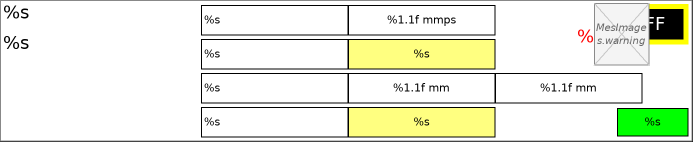
VISUALIZATION VISU_AXE_STD1_LIN_REL_FCT_ETAT_OSC  // 693x142
VAR_IN_OUT
	m_Input_MOTEUR: BLOCK_AXE_STD1_OSCILLANT;
	m_Input_PRG_MOUVEMENT_PS: BLOCK_PRG_MOUVEMENT_PS;
END_VAR
VAR_INPUT
	m_Input_ID_NOM_XML : INT;
END_VAR
    Rectangle (0,0 693x142), "%s", text list: 'TextList_Type_Moteur', text index: m_Input_ID_NOM_XML
    Rectangle (0,28 107x30), "%s", text variable: m_Input_MOTEUR.MNEMO
    RoundedRectangle (201,5 147x30), "%s", text list: 'TextList_Moteurs', text index: 7
    RoundedRectangle (201,39 147x30), "%s", text list: 'TextList_Moteurs', text index: 8
    RoundedRectangle (201,73 147x30), "%s", text list: 'TextList_Moteurs', text index: 9
    RoundedRectangle (201,107 147x30), "%s", text list: 'TextList_Moteurs', text index: 10
    RoundedRectangle (348,5 147x30), "%1.1f mmps", text variable: m_Input_MOTEUR.STATE_Vit
    RoundedRectangle (348,39 147x30), "%s", text variable: m_Input_MOTEUR.CONF_ID_POSTE[m_Input_MOTEUR.PRM_NPOSTE]
    RoundedRectangle (348,73 147x30), "%1.1f mm", text variable: m_Input_MOTEUR.STATE_Pos_Rel
    RoundedRectangle (495,73 147x30), "%1.1f mm", text variable: m_Input_MOTEUR.STATE_Pos
    RoundedRectangle (348,107 147x30), "%s", text variable: m_Input_MOTEUR.CONF_ID_REF[m_Input_MOTEUR.PRM_NRef]
    RoundedRectangle (617,108 71x28), "%s", invisible if: m_Input_MOTEUR.STATE_Homed OR m_Input_MOTEUR.CONF_No_Ref, text list: 'TextList_Moteurs', text index: 11
    RoundedRectangle (617,108 71x28), "%s", invisible if: NOT m_Input_MOTEUR.STATE_Homed OR m_Input_MOTEUR.CONF_No_Ref, text list: 'TextList_Moteurs', text index: 11
    RoundedRectangle (608,4 80x40), invisible if: NOT m_Input_MOTEUR.OP_Validation.OK
    RoundedRectangle (608,4 80x40), invisible if: NOT m_Input_MOTEUR.OP_Validation.AR
    RoundedRectangle (608,4 80x40), invisible if: NOT m_Input_MOTEUR.OP_Validation.EC
    RoundedRectangle (613,9 70x30), "ON", invisible if: m_Input_MOTEUR.STATE_Ar
    RoundedRectangle (613,9 70x30), "OFF", invisible if: NOT m_Input_MOTEUR.STATE_Ar
    Rectangle (535,24 67x21), "%i", text variable: m_Input_MOTEUR.STATE_Err, invisible if: NOT m_Input_MOTEUR.STATE_NOK
    Image (594,3 55x62), invisible if: NOT m_Input_MOTEUR.STATE_NOK, image: MesImages.warning
END_VISUALIZATION

(* stored: Version 1.1.0.1, ProductVersion 3.1.4024.10
   Visu VISU_AXE_STD1_LIN_REL_FCT_ETAT_OSC: Id {37a1f610-89bb-445e-87f5-660507e5b625} *)
